# EPICS substitutions: apps/richsimApp/Db/LVRICH1.substitutions
file "db/richlv_sim1.db" {
    pattern {HOST,CH,SCAN,PORT,DETALIAS}
  {"129.57.86.109",  "1","2 second","B_HW_LVRICH_CH0","B_DET_RICH_LV_CH0"}
  {"129.57.86.109",  "1","2 second","B_HW_LVRICH_CH1","B_DET_RICH_LV_CH1"}
  {"129.57.86.109",  "2","2 second","B_HW_LVRICH_CH2","B_DET_RICH_LV_CH2"}
  {"129.57.86.109",  "3","2 second","B_HW_LVRICH_CH3","B_DET_RICH_LV_CH3"}
  {"129.57.86.109",  "4","2 second","B_HW_LVRICH_CH4","B_DET_RICH_LV_CH4"}
  {"129.57.86.109",  "5","2 second","B_HW_LVRICH_CH5","B_DET_RICH_LV_CH5"}
  {"129.57.86.109",  "6","2 second","B_HW_LVRICH_CH6","B_DET_RICH_LV_CH6"}
  {"129.57.86.109",  "7","2 second","B_HW_LVRICH_CH7","B_DET_RICH_LV_CH7"}
  {"129.57.86.109",  "8","2 second","B_HW_LVRICH_CH8","B_DET_RICH_LV_CH8"}
  {"129.57.86.109",  "9","2 second","B_HW_LVRICH_CH9","B_DET_RICH_LV_CH9"}
  {"129.57.86.109",  "10","2 second","B_HW_LVRICH_CH10","B_DET_RICH_LV_CH10}
  {"129.57.86.109",  "11","2 second","B_HW_LVRICH_CH11","B_DET_RICH_LV_ch11"}
  {"129.57.86.109",  "12","2 second","B_HW_LVRICH_CH12","B_DET_RICH_LV_ch12"}
  {"129.57.86.109",  "13","2 second","B_HW_LVRICH_CH13","B_DET_RICH_LV_CH13"}
  {"129.57.86.109",  "14","2 second","B_HW_LVRICH_CH14","B_DET_RICH_LV_CH14"}
  {"129.57.86.109",  "15","2 second","B_HW_LVRICH_CH15","B_DET_RICH_LV_CH15"}
  {"129.57.86.109",  "16","2 second","B_HW_LVRICH_CH16","B_DET_RICH_LV_CH16"}
  {"129.57.86.109",  "17","2 second","B_HW_LVRICH_CH17","B_DET_RICH_LV_CH17"}
  {"129.57.86.109",  "18","2 second","B_HW_LVRICH_CH18","B_DET_RICH_LV_CH18"}
  {"129.57.86.109",  "19","2 second","B_HW_LVRICH_CH19","B_DET_RICH_LV_CH19"}
  {"129.57.86.109",  "20","2 second","B_HW_LVRICH_CH20","B_DET_RICH_LV_CH20"}
  {"129.57.86.109",  "21","2 second","B_HW_LVRICH_CH21","B_DET_RICH_LV_ch21"}
  {"129.57.86.109",  "22","2 second","B_HW_LVRICH_CH22","B_DET_RICH_LV_ch22"}
  {"129.57.86.109",  "23","2 second","B_HW_LVRICH_CH23","B_DET_RICH_LV_CH23"}
  {"129.57.86.109",  "24","2 second","B_HW_LVRICH_CH24","B_DET_RICH_LV_CH24"}
  {"129.57.86.109",  "25","2 second","B_HW_LVRICH_CH25","B_DET_RICH_LV_CH25"}
  {"129.57.86.109",  "26","2 second","B_HW_LVRICH_CH26","B_DET_RICH_LV_CH26"}
  {"129.57.86.109",  "27","2 second","B_HW_LVRICH_CH27","B_DET_RICH_LV_CH27"}
  {"129.57.86.109",  "28","2 second","B_HW_LVRICH_CH28","B_DET_RICH_LV_CH28"}
  {"129.57.86.109",  "29","2 second","B_HW_LVRICH_CH29","B_DET_RICH_LV_CH29"}
  {"129.57.86.109",  "30","2 second","B_HW_LVRICH_CH30","B_DET_RICH_LV_CH30"}
  {"129.57.86.109",  "31","2 second","B_HW_LVRICH_CH31","B_DET_RICH_LV_ch31"}
  {"129.57.86.109",  "32","2 second","B_HW_LVRICH_CH32","B_DET_RICH_LV_ch32"}
  {"129.57.86.109",  "33","2 second","B_HW_LVRICH_CH33","B_DET_RICH_LV_CH33"}
  {"129.57.86.109",  "34","2 second","B_HW_LVRICH_CH34","B_DET_RICH_LV_CH34"}
}
